# EPICS substitutions: FINS/FINS-IOC-01App/Db/sandals-gate-valve.substitutions
#
# Read addresses
#
# DM0000		Gate valve watchdog (increment from 1 to 255 every second)
# DM00001		V1 Gate valve status (reserved, not currently used)
# DM00002		V2 Gate valve status

global{TIMEOUT="\$(TIMEOUT=5.0)"}

file "$(TOP)/FINS-IOC-01App/Db/sandals-gate-valve.template" {
	{ P=\$(P), Q=\$(Q) }
}
